// TIA Portal V18 export
TYPE "UDT_AHUsSATSetPoints"
// stored: IsFailsafeCompliant false
   STRUCT
      Actual { S7_SetPoint := 'True'} : Array[1..3] of Real;
      Target : Array[1..3] of Real;
      MinAbs : Array[1..3] of Real;
      MaxAbs : Array[1..3] of Real;
   END_STRUCT;
END_TYPE
